{attribute addProperty BoxType "EL7201-0010-0030"}
{attribute addProperty Id "FB_PositionAT %I*FB_Position_BA8AA9F03240DRV_StatuswordAT %I*DRV_Statusword_53CBCECC1620DRV_ControlwordAT %Q*DRV_Controlword_417617681620DRV_Target_velocityAT %Q*DRV_Target_velocity_53A88AB03240WcStateAT %I*WcState_F855686C1620InfoDataAT %I*InfoData_81099714160200"}
{attribute addProperty CRC "490475478"}
{attribute addProperty SizeInBites "272"}
{attribute addProperty SizeInBytes "34"}
TYPE EL7201_F2E81963 :
STRUCT
	{attribute addProperty Name "FB_Position"}
	FB_Position : FB_Position_BA8AA9F0;
	{attribute addProperty Name "DRV_Statusword"}
	DRV_Statusword : DRV_Statusword_53CBCECC;
	{attribute addProperty Name "DRV_Controlword"}
	DRV_Controlword : DRV_Controlword_41761768;
	{attribute addProperty Name "DRV_Target_velocity"}
	DRV_Target_velocity : DRV_Target_velocity_53A88AB0;
	{attribute addProperty Name "WcState"}
	WcState : WcState_F855686C;
	{attribute addProperty Name "InfoData"}
	InfoData : InfoData_81099714;
END_STRUCT
END_TYPE

(* stored: Version 1.2.0.0, ProductVersion 3.1.4024.9
   DUT EL7201_F2E81963: Id {3b269101-f281-4f09-878e-63534b3d4942} *)
